{attribute addProperty BoxType "EK1100-0000-0018"}
{attribute addProperty Id "Beckhoff_EPP5xxxEK1122Beckhoff_EPP5xxxEK1122_A40EFD8E1568196"}
{attribute addProperty CRC "899269771"}
{attribute addProperty SizeInBites "1568"}
{attribute addProperty SizeInBytes "196"}
TYPE Beckhoff_EPP5xxx_3599C48B EXTENDS EK1100_179A0949 :
STRUCT
	{attribute addProperty Name "Beckhoff_EPP5xxxEK1122"}
	Beckhoff_EPP5xxxEK1122 : Beckhoff_EPP5xxxEK1122_A40EFD8E;
END_STRUCT
END_TYPE

(* stored: Version 1.2.0.0, ProductVersion 3.1.4024.9
   DUT Beckhoff_EPP5xxx_3599C48B: Id {0aa87a16-ca37-422f-ab23-a3d060c9f9ac} *)
